Universal Robots PolyScope program: kasi.urp

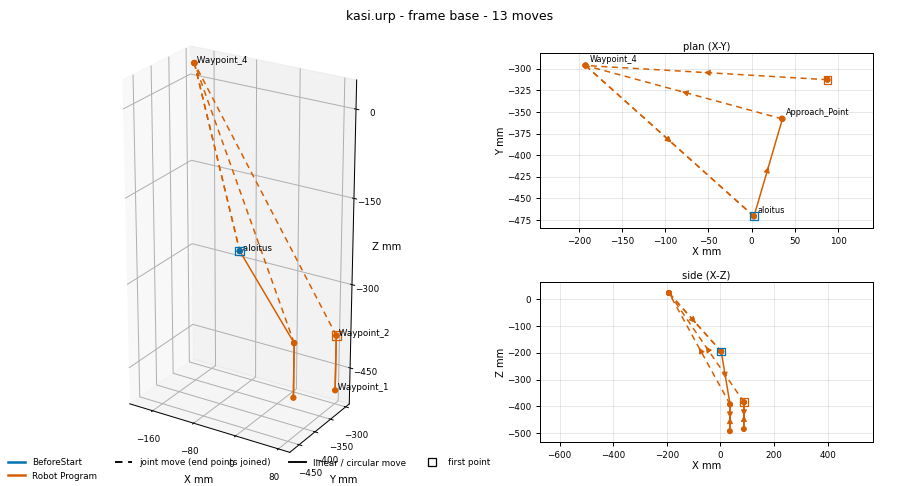
[picture p0: tool path of kasi.urp in frame base, 13 of 15 moves have a stored position in this frame; points joined in program order, loops and branches not executed]
Program kasi (installation=TVT17SPLAntti directory=/programs createdIn=3.10.0.76181 lastSavedIn=3.10.0.76181 robotSerialNumber=2018357902)
Calibrated DH parameters: a=[0.00015, -0.193406, -0.353214, 0.000101, 0.000049, 0]; d=[0.08934, 486.592682, -461.422552, -25.060198, 0.094902, 0.082419]; alpha=[1.570675, -0.000778, -0.00678, 1.570332, -1.570641, 0]; deltaTheta=[0.000035, -1.098336, 0.64827, 0.450067, -0.000055, 0.000056]
BeforeStart
  MoveJ speed 60 deg/s, acceleration 80 deg/s^2 (useActiveTCP=true)
    Waypoint aloitus: TCP in base x=2.713 y=-470.779 z=-194.927 mm, rx=0.0011 ry=-3.0383 rz=0.7917 rad; joints [288.818, -141.163, -140.572, 39.622, 81.192, 16.281] deg; flange x=2.963 y=-392.7 z=-55.272 mm, rx=0.0011 ry=-3.0383 rz=0.7917 rad
  mData := socket_open("192.168.100.11", 30000)
Robot Program (runOnlyOnce=false)
  SuppressedNode
    Loop Forever
      Wait Sleep waitTime=1
  Loop While (checkContinuously=false) expression=mData≟ False
    Wait Sleep waitTime=1
    mData := socket_open("192.168.100.11", 30000)
  kasky := socket_read_ascii_float(7)
  Loop While (checkContinuously=false) expression=kasky[0]≠7
    kasky := socket_read_ascii_float(7)
    Script: socket_send_string("O")
    Wait Sleep waitTime=1
  SuppressedNode
    Popup Message (haltProgram=false inputType=Variable) variable=kasky
  tuote := kasky[1]
  asento := [kasky[2], kasky[3], kasky[4], kasky[5], kasky[6], kasky[7]]
  If tuote≟0
    'Rectangle=0'
